INTERFACE IProcessSampleMover

METHOD GiveMover : IProcessSampleMover
VAR_INPUT
	mover : REFERENCE TO FB_Mover;
END_VAR
END_METHOD

(* % of completion of the process *)
PROPERTY iCompletionPC : INT
GET
END_GET
END_PROPERTY

PROPERTY Mover : REFERENCE TO FB_Mover
GET
END_GET
SET
END_SET
END_PROPERTY

PROPERTY ProcessExecution : ProcessExecution_e
GET
END_GET
SET
END_SET
END_PROPERTY

METHOD TakeMover : IProcessSampleMover
VAR_INPUT
END_VAR
END_METHOD

METHOD ToString : STRING
VAR_INPUT
END_VAR
END_METHOD

PROPERTY xBusy : BOOL
GET
END_GET
SET
END_SET
END_PROPERTY

PROPERTY xDone : BOOL
GET
END_GET
END_PROPERTY

PROPERTY xMoverPathFree : BOOL
GET
END_GET
END_PROPERTY

PROPERTY xMoverShouldLeave : BOOL
GET
END_GET
END_PROPERTY

END_INTERFACE

(* stored: Version 1.1.0.1, ProductVersion 3.1.4024.12
   Itf IProcessSampleMover: Id {e8a352f5-92c0-46fd-96c3-ad4169ca5226}
   Method GiveMover: Id {0a35138d-fff9-4cbb-bd80-60d414af24fe}
   Property iCompletionPC: Id {fbddfb68-6efd-4016-ab71-c8452d6f0a56}
   Get Get: Id {901c360f-2ab2-4960-8605-04aed755f357}
   Property Mover: Id {85439d31-f2ba-46f7-af41-2e3f2c528273}
   Get Get: Id {d22bd6ac-4638-4ff2-97cf-819eddbcf833}
   Set Set: Id {1f2d0179-eb69-4b55-b7c1-3e0fb48b780e}
   Property ProcessExecution: Id {e25fae5c-c258-4966-811f-ec988823a552}
   Get Get: Id {2f01004b-8a18-4b15-ab24-617de289448e}
   Set Set: Id {f1166bc6-2752-44af-bb31-b84aa09cee0c}
   Method TakeMover: Id {8cafca64-e16b-45c4-9368-909227c9595e}
   Method ToString: Id {6661c2c4-d4f5-4de9-b413-5f976e6e791f}
   Property xBusy: Id {7e4980be-98dc-4017-a605-db3726cae92d}
   Get Get: Id {0e18145d-7e25-4d5a-8397-8d55b3cf8467}
   Set Set: Id {5edc63b7-b2da-4efc-aa24-8c5a59b15482}
   Property xDone: Id {6e4f6236-7600-4370-bb3c-80c16f6a0227}
   Get Get: Id {7e4f205b-ea25-4f1f-ab24-0bfdf4b3290e}
   Property xMoverPathFree: Id {86f9f09e-e9cb-4cb5-bf79-76dc6d66f376}
   Get Get: Id {4f02ff20-871b-48b8-a1b4-856c0d28ee67}
   Property xMoverShouldLeave: Id {035b5043-bf81-4931-95a3-a90625d65048}
   Get Get: Id {ca578f10-e219-4084-92b9-a23e055801f2} *)
